Universal Robots PolyScope program: test3.urp

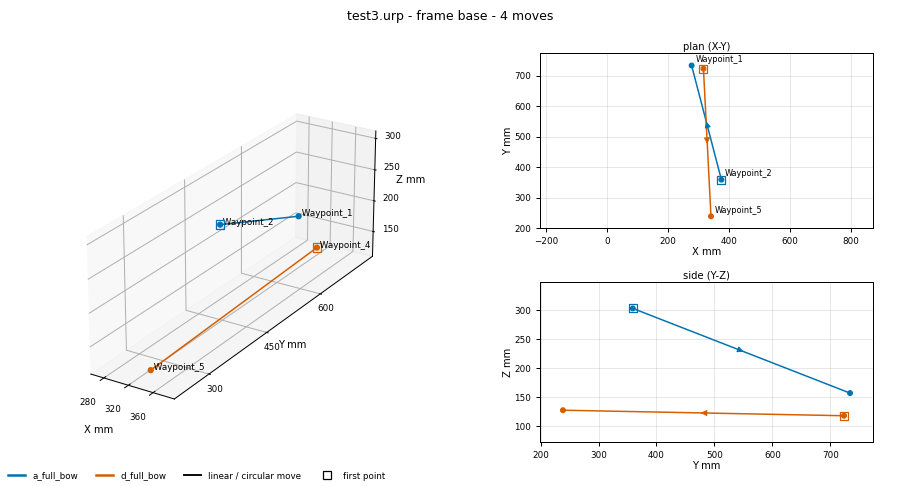
[picture p0: tool path of test3.urp in frame base, 4 of 7 moves have a stored position in this frame; points joined in program order, loops and branches not executed]
Program test3 (installation=string_planes directory=/programs createdIn=5.17.3 lastSavedIn=5.17.3 robotSerialNumber=20245501435)
Calibrated DH parameters: a=[0.000154, -0.137004, -0.385524, -0.00002, 0.000092, 0]; d=[0.162441, 211.794786, -230.585024, 18.923638, 0.099786, 0.09951]; alpha=[1.569493, -0.001902, 0.003874, 1.570111, -1.570167, 0]; deltaTheta=[0, -1.242934, 1.056292, 0.186646, 0.000002, 0.000001]
InitVariablesNode
Robot Program (runOnlyOnce=false)
  bow_section := -1
  Call a_full_bow
  Call a_to_d
  bow_dir := False
  Call d_full_bow
SubProgram -> d_full_bow
SubProgram -> a_to_d
SubProgram -> a_full_bow
SubProgram a_full_bow (keepSynchronizedWithDisk=false) programFile=/programs/a_full_bow.urp
  bow_dir := True
  note_dur := 1
  Timer (action=Start) variable(name=timer_1)
  If bow_dir
    MoveL speed 250 mm/s, acceleration 1200 mm/s^2 (useActiveTCP=true) feature=Base
      Waypoint Waypoint_2: TCP in base x=374.969 y=359.127 z=303.035 mm, rx=1.6275 ry=2.3373 rz=-1.1146 rad; joints [-156.117, -66.368, 101.552, -88.734, -114.429, -168.118] deg; TCP offset x=28.21 y=-96.107 z=-99.69 mm, rx=0 ry=0 rz=0 rad
        Until EXPRESSION (allowActions=false) ExpressionBranch=timer_1≟note_dur
  Else 
    MoveL speed 250 mm/s, acceleration 1200 mm/s^2 (useActiveTCP=true) feature=Base
      Waypoint Waypoint_1: TCP in base x=277.237 y=734.032 z=156.892 mm, rx=1.7389 ry=2.3104 rz=-1.1078 rad; joints [-126.647, -28.123, 54.729, -74.616, -91.964, -141.812] deg; TCP offset x=28.21 y=-96.107 z=-99.69 mm, rx=0 ry=0 rz=0 rad
        Until EXPRESSION (allowActions=false) ExpressionBranch=timer_1≟note_dur
  SuppressedNode
    MoveL speed 250 mm/s, acceleration 1200 mm/s^2 (useActiveTCP=true) feature=Base
      Waypoint Waypoint_1: TCP in base x=277.237 y=734.032 z=156.892 mm, rx=1.7389 ry=2.3104 rz=-1.1078 rad; joints [-126.647, -28.123, 54.729, -74.616, -91.964, -141.812] deg
      Waypoint Waypoint_3: motionParameters(blendRadius=0.05); TCP in base x=335.809 y=527.638 z=230.762 mm, rx=1.7389 ry=2.3104 rz=-1.1078 rad; joints [-141.244, -51.172, 87.867, -86.053, -101.589, -152.842] deg; TCP offset x=28.21 y=-96.107 z=-99.69 mm, rx=0 ry=0 rz=0 rad
      Waypoint Waypoint_2: TCP in base x=374.969 y=359.127 z=303.035 mm, rx=1.6275 ry=2.3373 rz=-1.1146 rad; joints [-156.117, -66.368, 101.552, -88.734, -114.429, -168.118] deg
  Timer (action=Stop) variable=timer_1
  Timer (action=Reset) variable=timer_1
SubProgram a_to_d (keepSynchronizedWithDisk=false) programFile=/programs/string_crossings/a_to_d.urp
  If bow_section≟-1
    MoveJ speed 60 deg/s, acceleration 80 deg/s^2 (useActiveTCP=true) feature=Base
      Waypoint Waypoint_9 (Relative): relativeFromPosition TCP in base x=277.235 y=734.032 z=156.893 mm, rx=1.7389 ry=2.3104 rz=-1.1077 rad; joints [-126.647, -28.124, 54.729, -74.617, -91.964, -141.812] deg; TCP in base x=340.806 y=238.633 z=127.349 mm, rx=-1.5375 ry=-2.1223 rz=1.0863 rad; joints [-167.853, -53.47, 123.567, -113.68, -104.543, -179.466] deg
  ElseIf bow_section≟0
    MoveJ speed 60 deg/s, acceleration 80 deg/s^2 (useActiveTCP=true) feature=Base
      Waypoint Waypoint_9 (Relative): relativeFromPosition TCP in base x=277.235 y=734.032 z=156.893 mm, rx=1.7389 ry=2.3104 rz=-1.1077 rad; joints [-126.647, -28.124, 54.729, -74.617, -91.964, -141.812] deg; TCP in base x=340.806 y=238.633 z=127.349 mm, rx=-1.5375 ry=-2.1223 rz=1.0863 rad; joints [-167.853, -53.47, 123.567, -113.68, -104.543, -179.466] deg
  Else 
    MoveJ speed 60 deg/s, acceleration 80 deg/s^2 (useActiveTCP=true) feature=Base
      Waypoint Waypoint_9 (Relative): relativeFromPosition TCP in base x=277.235 y=734.032 z=156.893 mm, rx=1.7389 ry=2.3104 rz=-1.1077 rad; joints [-126.647, -28.124, 54.729, -74.617, -91.964, -141.812] deg; TCP in base x=340.806 y=238.633 z=127.349 mm, rx=-1.5375 ry=-2.1223 rz=1.0863 rad; joints [-167.853, -53.47, 123.567, -113.68, -104.543, -179.466] deg
SubProgram d_full_bow (keepSynchronizedWithDisk=false) programFile=/programs/d_full_bow.urp
  bow_dir := True
  note_dur := 1
  Timer (action=Start) variable=timer_1
  If bow_dir≟ False
    MoveL speed 250 mm/s, acceleration 1200 mm/s^2 (useActiveTCP=true) feature=Base
      Waypoint Waypoint_4: TCP in base x=316.077 y=723.624 z=117.8 mm, rx=-1.5349 ry=-2.2386 rz=1.1274 rad; joints [-128.458, -21.868, 50.818, -72.931, -81.953, -152.853] deg
        Until EXPRESSION (allowActions=false) ExpressionBranch=timer_1≟note_dur
  Else 
    MoveL speed 250 mm/s, acceleration 1200 mm/s^2 (useActiveTCP=true) feature=Base
      Waypoint Waypoint_5: TCP in base x=340.806 y=238.625 z=127.338 mm, rx=-1.5375 ry=-2.1223 rz=1.0863 rad; joints [-167.854, -53.469, 123.568, -113.681, -104.543, -179.466] deg
        Until EXPRESSION (allowActions=false) ExpressionBranch=timer_1≟note_dur
  SuppressedNode
    MoveL speed 250 mm/s, acceleration 1200 mm/s^2 (useActiveTCP=true) feature=Base
      Waypoint Waypoint_1: TCP in base x=331.973 y=720.894 z=108.291 mm, rx=-1.645 ry=-2.1081 rz=1.0591 rad; joints [-129.773, -21.651, 52.373, -76.468, -76.907, -149.022] deg
      Waypoint Waypoint_2: motionParameters(blendRadius=0.05); TCP in base x=332.259 y=481.199 z=108.291 mm, rx=-1.645 ry=-2.1081 rz=1.0591 rad; joints [-144.031, -41.816, 97.865, -100.392, -86.961, -159.136] deg
      Waypoint Waypoint_3: TCP in base x=332.566 y=223.853 z=108.291 mm, rx=-1.645 ry=-2.1081 rz=1.0591 rad; joints [-170.229, -51.627, 126.122, -120.942, -105.516, -177.767] deg
  Timer (action=Stop) variable=timer_1
  Timer (action=Reset) variable=timer_1
